// TIA Portal V15.1 export
// export: Created 2020-12-28T13:40:55.3097416Z, ExportSetting WithDefaults, WithReadOnly, DisplayName Totally Integrated Automation Portal, DisplayVersion V15.1 Update 3, DisplayName TIA Portal Openness, DisplayVersion V15.1, DisplayName STEP 7 Professional, DisplayVersion V15.1 Update 3, DisplayName WinCC Advanced, DisplayVersion V15.1 Update 3
DATA_BLOCK "INST TBL TABLE LH"   // DB900
{ S7_Optimized_Access := 'TRUE' }
VERSION : 0.1
// stored: AutoNumber false, CodeModifiedDate 2020-12-28T13:20:36.0178679Z, CompileDate 2020-12-28T13:40:46.9815401Z, CreationDate 2020-12-28T13:20:35.8743592Z, DBAccessibleFromOPCUA true, DownloadWithoutReinit false, InstanceOfName 3STATE_PISTON, InstanceOfNumber 1101, InstanceOfType FB, InterfaceModifiedDate 2020-12-10T07:03:04.0661374Z, IsConsistent true, IsKnowHowProtected false, IsRetainMemResEnabled false, MemoryReserve 100, ModifiedDate 2020-12-28T13:20:36.0178679Z, ParameterModified 2020-12-10T07:03:04.0661374Z, StructureModified 2020-12-10T07:03:04.0661374Z, UDAEnableTagReadback false
"3STATE_PISTON"
   // VAR_INPUT
   //    in_safety : Bool;
   //    in_move_hp : Bool;
   //    in_move_wp : Bool;
   //    in_move_idle : Bool;
   //    in_sensor_hp : Bool;
   //    in_sensor_wp : Bool;
   // END_VAR
   // VAR_OUTPUT
   //    out_in_hp : Bool;
   //    out_in_wp : Bool;
   //    out_idle : Bool;
   //    out_status : Int;
   // END_VAR
   // VAR_IN_OUT
   //    in_ez_hp : Bool;
   //    in_ez_wp : Bool;
   //    in_ez_idle : Bool;
   // END_VAR
   // VAR
   //    "time" : Time;
   //    T : Struct
   //       tt1 : IEC_TIMER;
   //       tt2_hp { S7_SetPoint := 'True'} : IEC_TIMER;
   //       tt3_wp { S7_SetPoint := 'True'} : IEC_TIMER;
   //    END_STRUCT;
   // END_VAR
BEGIN
END_DATA_BLOCK

DATA_BLOCK "INST TBL TABLE RH"   // DB901
{ S7_Optimized_Access := 'TRUE' }
VERSION : 0.1
// stored: AutoNumber false, CodeModifiedDate 2020-12-28T13:20:36.0178679Z, CompileDate 2020-12-28T13:40:46.9815401Z, CreationDate 2020-12-28T13:20:35.8743592Z, DBAccessibleFromOPCUA true, DownloadWithoutReinit false, InstanceOfName 3STATE_PISTON, InstanceOfNumber 1101, InstanceOfType FB, InterfaceModifiedDate 2020-12-10T07:03:04.0661374Z, IsConsistent true, IsKnowHowProtected false, IsRetainMemResEnabled false, MemoryReserve 100, ModifiedDate 2020-12-28T13:20:36.0178679Z, ParameterModified 2020-12-10T07:03:04.0661374Z, StructureModified 2020-12-10T07:03:04.0661374Z, UDAEnableTagReadback false
"3STATE_PISTON"
   // VAR_INPUT
   //    in_safety : Bool;
   //    in_move_hp : Bool;
   //    in_move_wp : Bool;
   //    in_move_idle : Bool;
   //    in_sensor_hp : Bool;
   //    in_sensor_wp : Bool;
   // END_VAR
   // VAR_OUTPUT
   //    out_in_hp : Bool;
   //    out_in_wp : Bool;
   //    out_idle : Bool;
   //    out_status : Int;
   // END_VAR
   // VAR_IN_OUT
   //    in_ez_hp : Bool;
   //    in_ez_wp : Bool;
   //    in_ez_idle : Bool;
   // END_VAR
   // VAR
   //    "time" : Time;
   //    T : Struct
   //       tt1 : IEC_TIMER;
   //       tt2_hp { S7_SetPoint := 'True'} : IEC_TIMER;
   //       tt3_wp { S7_SetPoint := 'True'} : IEC_TIMER;
   //    END_STRUCT;
   // END_VAR
BEGIN
END_DATA_BLOCK

DATA_BLOCK "INST TBL SECTION1"   // DB902
{ S7_Optimized_Access := 'TRUE' }
VERSION : 0.1
// stored: AutoNumber false, CodeModifiedDate 2020-12-28T13:20:36.0178679Z, CompileDate 2020-12-28T13:40:46.9815401Z, CreationDate 2020-12-28T13:20:35.8743592Z, DBAccessibleFromOPCUA true, DownloadWithoutReinit false, InstanceOfName 3STATE_PISTON, InstanceOfNumber 1101, InstanceOfType FB, InterfaceModifiedDate 2020-12-10T07:03:04.0661374Z, IsConsistent true, IsKnowHowProtected false, IsRetainMemResEnabled false, MemoryReserve 100, ModifiedDate 2020-12-28T13:20:36.0178679Z, ParameterModified 2020-12-10T07:03:04.0661374Z, StructureModified 2020-12-10T07:03:04.0661374Z, UDAEnableTagReadback false
"3STATE_PISTON"
   // VAR_INPUT
   //    in_safety : Bool;
   //    in_move_hp : Bool;
   //    in_move_wp : Bool;
   //    in_move_idle : Bool;
   //    in_sensor_hp : Bool;
   //    in_sensor_wp : Bool;
   // END_VAR
   // VAR_OUTPUT
   //    out_in_hp : Bool;
   //    out_in_wp : Bool;
   //    out_idle : Bool;
   //    out_status : Int;
   // END_VAR
   // VAR_IN_OUT
   //    in_ez_hp : Bool;
   //    in_ez_wp : Bool;
   //    in_ez_idle : Bool;
   // END_VAR
   // VAR
   //    "time" : Time;
   //    T : Struct
   //       tt1 : IEC_TIMER;
   //       tt2_hp { S7_SetPoint := 'True'} : IEC_TIMER;
   //       tt3_wp { S7_SetPoint := 'True'} : IEC_TIMER;
   //    END_STRUCT;
   // END_VAR
BEGIN
END_DATA_BLOCK

DATA_BLOCK "INST TBL SECTION2"   // DB903
{ S7_Optimized_Access := 'TRUE' }
VERSION : 0.1
// stored: AutoNumber false, CodeModifiedDate 2020-12-28T13:20:36.0178679Z, CompileDate 2020-12-28T13:40:46.9815401Z, CreationDate 2020-12-28T13:20:35.8743592Z, DBAccessibleFromOPCUA true, DownloadWithoutReinit false, InstanceOfName 3STATE_PISTON, InstanceOfNumber 1101, InstanceOfType FB, InterfaceModifiedDate 2020-12-10T07:03:04.0661374Z, IsConsistent true, IsKnowHowProtected false, IsRetainMemResEnabled false, MemoryReserve 100, ModifiedDate 2020-12-28T13:20:36.0178679Z, ParameterModified 2020-12-10T07:03:04.0661374Z, StructureModified 2020-12-10T07:03:04.0661374Z, UDAEnableTagReadback false
"3STATE_PISTON"
   // VAR_INPUT
   //    in_safety : Bool;
   //    in_move_hp : Bool;
   //    in_move_wp : Bool;
   //    in_move_idle : Bool;
   //    in_sensor_hp : Bool;
   //    in_sensor_wp : Bool;
   // END_VAR
   // VAR_OUTPUT
   //    out_in_hp : Bool;
   //    out_in_wp : Bool;
   //    out_idle : Bool;
   //    out_status : Int;
   // END_VAR
   // VAR_IN_OUT
   //    in_ez_hp : Bool;
   //    in_ez_wp : Bool;
   //    in_ez_idle : Bool;
   // END_VAR
   // VAR
   //    "time" : Time;
   //    T : Struct
   //       tt1 : IEC_TIMER;
   //       tt2_hp { S7_SetPoint := 'True'} : IEC_TIMER;
   //       tt3_wp { S7_SetPoint := 'True'} : IEC_TIMER;
   //    END_STRUCT;
   // END_VAR
BEGIN
END_DATA_BLOCK

DATA_BLOCK "INST TBL SECTION4 LH"   // DB904
{ S7_Optimized_Access := 'TRUE' }
VERSION : 0.1
// stored: AutoNumber false, CodeModifiedDate 2020-12-28T13:20:36.0178679Z, CompileDate 2020-12-28T13:40:46.9815401Z, CreationDate 2020-12-28T13:20:35.8743592Z, DBAccessibleFromOPCUA true, DownloadWithoutReinit false, InstanceOfName 3STATE_PISTON, InstanceOfNumber 1101, InstanceOfType FB, InterfaceModifiedDate 2020-12-10T07:03:04.0661374Z, IsConsistent true, IsKnowHowProtected false, IsRetainMemResEnabled false, MemoryReserve 100, ModifiedDate 2020-12-28T13:20:36.0178679Z, ParameterModified 2020-12-10T07:03:04.0661374Z, StructureModified 2020-12-10T07:03:04.0661374Z, UDAEnableTagReadback false
"3STATE_PISTON"
   // VAR_INPUT
   //    in_safety : Bool;
   //    in_move_hp : Bool;
   //    in_move_wp : Bool;
   //    in_move_idle : Bool;
   //    in_sensor_hp : Bool;
   //    in_sensor_wp : Bool;
   // END_VAR
   // VAR_OUTPUT
   //    out_in_hp : Bool;
   //    out_in_wp : Bool;
   //    out_idle : Bool;
   //    out_status : Int;
   // END_VAR
   // VAR_IN_OUT
   //    in_ez_hp : Bool;
   //    in_ez_wp : Bool;
   //    in_ez_idle : Bool;
   // END_VAR
   // VAR
   //    "time" : Time;
   //    T : Struct
   //       tt1 : IEC_TIMER;
   //       tt2_hp { S7_SetPoint := 'True'} : IEC_TIMER;
   //       tt3_wp { S7_SetPoint := 'True'} : IEC_TIMER;
   //    END_STRUCT;
   // END_VAR
BEGIN
END_DATA_BLOCK

DATA_BLOCK "INST TBL SECTION4 RH"   // DB905
{ S7_Optimized_Access := 'TRUE' }
VERSION : 0.1
// stored: AutoNumber false, CodeModifiedDate 2020-12-28T13:20:36.0178679Z, CompileDate 2020-12-28T13:40:46.9815401Z, CreationDate 2020-12-28T13:20:35.8743592Z, DBAccessibleFromOPCUA true, DownloadWithoutReinit false, InstanceOfName 3STATE_PISTON, InstanceOfNumber 1101, InstanceOfType FB, InterfaceModifiedDate 2020-12-10T07:03:04.0661374Z, IsConsistent true, IsKnowHowProtected false, IsRetainMemResEnabled false, MemoryReserve 100, ModifiedDate 2020-12-28T13:20:36.0178679Z, ParameterModified 2020-12-10T07:03:04.0661374Z, StructureModified 2020-12-10T07:03:04.0661374Z, UDAEnableTagReadback false
"3STATE_PISTON"
   // VAR_INPUT
   //    in_safety : Bool;
   //    in_move_hp : Bool;
   //    in_move_wp : Bool;
   //    in_move_idle : Bool;
   //    in_sensor_hp : Bool;
   //    in_sensor_wp : Bool;
   // END_VAR
   // VAR_OUTPUT
   //    out_in_hp : Bool;
   //    out_in_wp : Bool;
   //    out_idle : Bool;
   //    out_status : Int;
   // END_VAR
   // VAR_IN_OUT
   //    in_ez_hp : Bool;
   //    in_ez_wp : Bool;
   //    in_ez_idle : Bool;
   // END_VAR
   // VAR
   //    "time" : Time;
   //    T : Struct
   //       tt1 : IEC_TIMER;
   //       tt2_hp { S7_SetPoint := 'True'} : IEC_TIMER;
   //       tt3_wp { S7_SetPoint := 'True'} : IEC_TIMER;
   //    END_STRUCT;
   // END_VAR
BEGIN
END_DATA_BLOCK

DATA_BLOCK "INST TBL SECTION5 LH"   // DB906
{ S7_Optimized_Access := 'TRUE' }
VERSION : 0.1
// stored: AutoNumber false, CodeModifiedDate 2020-12-28T13:20:36.0178679Z, CompileDate 2020-12-28T13:40:46.9815401Z, CreationDate 2020-12-28T13:20:35.8743592Z, DBAccessibleFromOPCUA true, DownloadWithoutReinit false, InstanceOfName 3STATE_PISTON, InstanceOfNumber 1101, InstanceOfType FB, InterfaceModifiedDate 2020-12-10T07:03:04.0661374Z, IsConsistent true, IsKnowHowProtected false, IsRetainMemResEnabled false, MemoryReserve 100, ModifiedDate 2020-12-28T13:20:36.0178679Z, ParameterModified 2020-12-10T07:03:04.0661374Z, StructureModified 2020-12-10T07:03:04.0661374Z, UDAEnableTagReadback false
"3STATE_PISTON"
   // VAR_INPUT
   //    in_safety : Bool;
   //    in_move_hp : Bool;
   //    in_move_wp : Bool;
   //    in_move_idle : Bool;
   //    in_sensor_hp : Bool;
   //    in_sensor_wp : Bool;
   // END_VAR
   // VAR_OUTPUT
   //    out_in_hp : Bool;
   //    out_in_wp : Bool;
   //    out_idle : Bool;
   //    out_status : Int;
   // END_VAR
   // VAR_IN_OUT
   //    in_ez_hp : Bool;
   //    in_ez_wp : Bool;
   //    in_ez_idle : Bool;
   // END_VAR
   // VAR
   //    "time" : Time;
   //    T : Struct
   //       tt1 : IEC_TIMER;
   //       tt2_hp { S7_SetPoint := 'True'} : IEC_TIMER;
   //       tt3_wp { S7_SetPoint := 'True'} : IEC_TIMER;
   //    END_STRUCT;
   // END_VAR
BEGIN
END_DATA_BLOCK

DATA_BLOCK "INST TBL SECTION5 RH"   // DB907
{ S7_Optimized_Access := 'TRUE' }
VERSION : 0.1
// stored: AutoNumber false, CodeModifiedDate 2020-12-28T13:20:36.0178679Z, CompileDate 2020-12-28T13:40:46.9815401Z, CreationDate 2020-12-28T13:20:35.8743592Z, DBAccessibleFromOPCUA true, DownloadWithoutReinit false, InstanceOfName 3STATE_PISTON, InstanceOfNumber 1101, InstanceOfType FB, InterfaceModifiedDate 2020-12-10T07:03:04.0661374Z, IsConsistent true, IsKnowHowProtected false, IsRetainMemResEnabled false, MemoryReserve 100, ModifiedDate 2020-12-28T13:20:36.0178679Z, ParameterModified 2020-12-10T07:03:04.0661374Z, StructureModified 2020-12-10T07:03:04.0661374Z, UDAEnableTagReadback false
"3STATE_PISTON"
   // VAR_INPUT
   //    in_safety : Bool;
   //    in_move_hp : Bool;
   //    in_move_wp : Bool;
   //    in_move_idle : Bool;
   //    in_sensor_hp : Bool;
   //    in_sensor_wp : Bool;
   // END_VAR
   // VAR_OUTPUT
   //    out_in_hp : Bool;
   //    out_in_wp : Bool;
   //    out_idle : Bool;
   //    out_status : Int;
   // END_VAR
   // VAR_IN_OUT
   //    in_ez_hp : Bool;
   //    in_ez_wp : Bool;
   //    in_ez_idle : Bool;
   // END_VAR
   // VAR
   //    "time" : Time;
   //    T : Struct
   //       tt1 : IEC_TIMER;
   //       tt2_hp { S7_SetPoint := 'True'} : IEC_TIMER;
   //       tt3_wp { S7_SetPoint := 'True'} : IEC_TIMER;
   //    END_STRUCT;
   // END_VAR
BEGIN
END_DATA_BLOCK

DATA_BLOCK "INST TBL POSITIONING LH"   // DB908
{ S7_Optimized_Access := 'TRUE' }
VERSION : 0.1
// stored: AutoNumber false, CodeModifiedDate 2020-12-28T13:20:36.0178679Z, CompileDate 2020-12-28T13:40:46.9815401Z, CreationDate 2020-12-28T13:20:35.8743592Z, DBAccessibleFromOPCUA true, DownloadWithoutReinit false, InstanceOfName 3STATE_PISTON, InstanceOfNumber 1101, InstanceOfType FB, InterfaceModifiedDate 2020-12-10T07:03:04.0661374Z, IsConsistent true, IsKnowHowProtected false, IsRetainMemResEnabled false, MemoryReserve 100, ModifiedDate 2020-12-28T13:20:36.0178679Z, ParameterModified 2020-12-10T07:03:04.0661374Z, StructureModified 2020-12-10T07:03:04.0661374Z, UDAEnableTagReadback false
"3STATE_PISTON"
   // VAR_INPUT
   //    in_safety : Bool;
   //    in_move_hp : Bool;
   //    in_move_wp : Bool;
   //    in_move_idle : Bool;
   //    in_sensor_hp : Bool;
   //    in_sensor_wp : Bool;
   // END_VAR
   // VAR_OUTPUT
   //    out_in_hp : Bool;
   //    out_in_wp : Bool;
   //    out_idle : Bool;
   //    out_status : Int;
   // END_VAR
   // VAR_IN_OUT
   //    in_ez_hp : Bool;
   //    in_ez_wp : Bool;
   //    in_ez_idle : Bool;
   // END_VAR
   // VAR
   //    "time" : Time;
   //    T : Struct
   //       tt1 : IEC_TIMER;
   //       tt2_hp { S7_SetPoint := 'True'} : IEC_TIMER;
   //       tt3_wp { S7_SetPoint := 'True'} : IEC_TIMER;
   //    END_STRUCT;
   // END_VAR
BEGIN
END_DATA_BLOCK

DATA_BLOCK "INST TBL POSITIONING RH"   // DB909
{ S7_Optimized_Access := 'TRUE' }
VERSION : 0.1
// stored: AutoNumber false, CodeModifiedDate 2020-12-28T13:20:36.0178679Z, CompileDate 2020-12-28T13:40:46.9815401Z, CreationDate 2020-12-28T13:20:35.8743592Z, DBAccessibleFromOPCUA true, DownloadWithoutReinit false, InstanceOfName 3STATE_PISTON, InstanceOfNumber 1101, InstanceOfType FB, InterfaceModifiedDate 2020-12-10T07:03:04.0661374Z, IsConsistent true, IsKnowHowProtected false, IsRetainMemResEnabled false, MemoryReserve 100, ModifiedDate 2020-12-28T13:20:36.0178679Z, ParameterModified 2020-12-10T07:03:04.0661374Z, StructureModified 2020-12-10T07:03:04.0661374Z, UDAEnableTagReadback false
"3STATE_PISTON"
   // VAR_INPUT
   //    in_safety : Bool;
   //    in_move_hp : Bool;
   //    in_move_wp : Bool;
   //    in_move_idle : Bool;
   //    in_sensor_hp : Bool;
   //    in_sensor_wp : Bool;
   // END_VAR
   // VAR_OUTPUT
   //    out_in_hp : Bool;
   //    out_in_wp : Bool;
   //    out_idle : Bool;
   //    out_status : Int;
   // END_VAR
   // VAR_IN_OUT
   //    in_ez_hp : Bool;
   //    in_ez_wp : Bool;
   //    in_ez_idle : Bool;
   // END_VAR
   // VAR
   //    "time" : Time;
   //    T : Struct
   //       tt1 : IEC_TIMER;
   //       tt2_hp { S7_SetPoint := 'True'} : IEC_TIMER;
   //       tt3_wp { S7_SetPoint := 'True'} : IEC_TIMER;
   //    END_STRUCT;
   // END_VAR
BEGIN
END_DATA_BLOCK

DATA_BLOCK "INST TBL PIN LH"   // DB910
{ S7_Optimized_Access := 'TRUE' }
VERSION : 0.1
// stored: AutoNumber false, CodeModifiedDate 2020-12-28T13:20:36.0178679Z, CompileDate 2020-12-28T13:40:46.9815401Z, CreationDate 2020-12-28T13:20:35.8743592Z, DBAccessibleFromOPCUA true, DownloadWithoutReinit false, InstanceOfName 3STATE_PISTON, InstanceOfNumber 1101, InstanceOfType FB, InterfaceModifiedDate 2020-12-10T07:03:04.0661374Z, IsConsistent true, IsKnowHowProtected false, IsRetainMemResEnabled false, MemoryReserve 100, ModifiedDate 2020-12-28T13:20:36.0178679Z, ParameterModified 2020-12-10T07:03:04.0661374Z, StructureModified 2020-12-10T07:03:04.0661374Z, UDAEnableTagReadback false
"3STATE_PISTON"
   // VAR_INPUT
   //    in_safety : Bool;
   //    in_move_hp : Bool;
   //    in_move_wp : Bool;
   //    in_move_idle : Bool;
   //    in_sensor_hp : Bool;
   //    in_sensor_wp : Bool;
   // END_VAR
   // VAR_OUTPUT
   //    out_in_hp : Bool;
   //    out_in_wp : Bool;
   //    out_idle : Bool;
   //    out_status : Int;
   // END_VAR
   // VAR_IN_OUT
   //    in_ez_hp : Bool;
   //    in_ez_wp : Bool;
   //    in_ez_idle : Bool;
   // END_VAR
   // VAR
   //    "time" : Time;
   //    T : Struct
   //       tt1 : IEC_TIMER;
   //       tt2_hp { S7_SetPoint := 'True'} : IEC_TIMER;
   //       tt3_wp { S7_SetPoint := 'True'} : IEC_TIMER;
   //    END_STRUCT;
   // END_VAR
BEGIN
END_DATA_BLOCK

DATA_BLOCK "INST TBL PIN RH"   // DB911
{ S7_Optimized_Access := 'TRUE' }
VERSION : 0.1
// stored: AutoNumber false, CodeModifiedDate 2020-12-28T13:20:36.0178679Z, CompileDate 2020-12-28T13:40:46.9815401Z, CreationDate 2020-12-28T13:20:35.8743592Z, DBAccessibleFromOPCUA true, DownloadWithoutReinit false, InstanceOfName 3STATE_PISTON, InstanceOfNumber 1101, InstanceOfType FB, InterfaceModifiedDate 2020-12-10T07:03:04.0661374Z, IsConsistent true, IsKnowHowProtected false, IsRetainMemResEnabled false, MemoryReserve 100, ModifiedDate 2020-12-28T13:20:36.0178679Z, ParameterModified 2020-12-10T07:03:04.0661374Z, StructureModified 2020-12-10T07:03:04.0661374Z, UDAEnableTagReadback false
"3STATE_PISTON"
   // VAR_INPUT
   //    in_safety : Bool;
   //    in_move_hp : Bool;
   //    in_move_wp : Bool;
   //    in_move_idle : Bool;
   //    in_sensor_hp : Bool;
   //    in_sensor_wp : Bool;
   // END_VAR
   // VAR_OUTPUT
   //    out_in_hp : Bool;
   //    out_in_wp : Bool;
   //    out_idle : Bool;
   //    out_status : Int;
   // END_VAR
   // VAR_IN_OUT
   //    in_ez_hp : Bool;
   //    in_ez_wp : Bool;
   //    in_ez_idle : Bool;
   // END_VAR
   // VAR
   //    "time" : Time;
   //    T : Struct
   //       tt1 : IEC_TIMER;
   //       tt2_hp { S7_SetPoint := 'True'} : IEC_TIMER;
   //       tt3_wp { S7_SetPoint := 'True'} : IEC_TIMER;
   //    END_STRUCT;
   // END_VAR
BEGIN
END_DATA_BLOCK

DATA_BLOCK "INST TBL SCREW GRIPPER"   // DB912
{ S7_Optimized_Access := 'TRUE' }
VERSION : 0.1
// stored: AutoNumber false, CodeModifiedDate 2020-12-28T13:20:36.0178679Z, CompileDate 2020-12-28T13:40:46.9815401Z, CreationDate 2020-12-28T13:20:35.8743592Z, DBAccessibleFromOPCUA true, DownloadWithoutReinit false, InstanceOfName 3STATE_PISTON, InstanceOfNumber 1101, InstanceOfType FB, InterfaceModifiedDate 2020-12-10T07:03:04.0661374Z, IsConsistent true, IsKnowHowProtected false, IsRetainMemResEnabled false, MemoryReserve 100, ModifiedDate 2020-12-28T13:20:36.0178679Z, ParameterModified 2020-12-10T07:03:04.0661374Z, StructureModified 2020-12-10T07:03:04.0661374Z, UDAEnableTagReadback false
"3STATE_PISTON"
   // VAR_INPUT
   //    in_safety : Bool;
   //    in_move_hp : Bool;
   //    in_move_wp : Bool;
   //    in_move_idle : Bool;
   //    in_sensor_hp : Bool;
   //    in_sensor_wp : Bool;
   // END_VAR
   // VAR_OUTPUT
   //    out_in_hp : Bool;
   //    out_in_wp : Bool;
   //    out_idle : Bool;
   //    out_status : Int;
   // END_VAR
   // VAR_IN_OUT
   //    in_ez_hp : Bool;
   //    in_ez_wp : Bool;
   //    in_ez_idle : Bool;
   // END_VAR
   // VAR
   //    "time" : Time;
   //    T : Struct
   //       tt1 : IEC_TIMER;
   //       tt2_hp { S7_SetPoint := 'True'} : IEC_TIMER;
   //       tt3_wp { S7_SetPoint := 'True'} : IEC_TIMER;
   //    END_STRUCT;
   // END_VAR
BEGIN
END_DATA_BLOCK

DATA_BLOCK "INST TBL WRAP GRIPPER"   // DB913
{ S7_Optimized_Access := 'TRUE' }
VERSION : 0.1
// stored: AutoNumber false, CodeModifiedDate 2020-12-28T13:20:36.0178679Z, CompileDate 2020-12-28T13:40:46.9815401Z, CreationDate 2020-12-28T13:20:35.8743592Z, DBAccessibleFromOPCUA true, DownloadWithoutReinit false, InstanceOfName 3STATE_PISTON, InstanceOfNumber 1101, InstanceOfType FB, InterfaceModifiedDate 2020-12-10T07:03:04.0661374Z, IsConsistent true, IsKnowHowProtected false, IsRetainMemResEnabled false, MemoryReserve 100, ModifiedDate 2020-12-28T13:20:36.0178679Z, ParameterModified 2020-12-10T07:03:04.0661374Z, StructureModified 2020-12-10T07:03:04.0661374Z, UDAEnableTagReadback false
"3STATE_PISTON"
   // VAR_INPUT
   //    in_safety : Bool;
   //    in_move_hp : Bool;
   //    in_move_wp : Bool;
   //    in_move_idle : Bool;
   //    in_sensor_hp : Bool;
   //    in_sensor_wp : Bool;
   // END_VAR
   // VAR_OUTPUT
   //    out_in_hp : Bool;
   //    out_in_wp : Bool;
   //    out_idle : Bool;
   //    out_status : Int;
   // END_VAR
   // VAR_IN_OUT
   //    in_ez_hp : Bool;
   //    in_ez_wp : Bool;
   //    in_ez_idle : Bool;
   // END_VAR
   // VAR
   //    "time" : Time;
   //    T : Struct
   //       tt1 : IEC_TIMER;
   //       tt2_hp { S7_SetPoint := 'True'} : IEC_TIMER;
   //       tt3_wp { S7_SetPoint := 'True'} : IEC_TIMER;
   //    END_STRUCT;
   // END_VAR
BEGIN
END_DATA_BLOCK

DATA_BLOCK "INST ST1 POSITIONING"   // DB914
{ S7_Optimized_Access := 'TRUE' }
VERSION : 0.1
// stored: AutoNumber false, CodeModifiedDate 2020-12-28T13:20:36.0178679Z, CompileDate 2020-12-28T13:40:46.9815401Z, CreationDate 2020-12-28T13:20:35.8743592Z, DBAccessibleFromOPCUA true, DownloadWithoutReinit false, InstanceOfName 3STATE_PISTON, InstanceOfNumber 1101, InstanceOfType FB, InterfaceModifiedDate 2020-12-10T07:03:04.0661374Z, IsConsistent true, IsKnowHowProtected false, IsRetainMemResEnabled false, MemoryReserve 100, ModifiedDate 2020-12-28T13:20:36.0178679Z, ParameterModified 2020-12-10T07:03:04.0661374Z, StructureModified 2020-12-10T07:03:04.0661374Z, UDAEnableTagReadback false
"3STATE_PISTON"
   // VAR_INPUT
   //    in_safety : Bool;
   //    in_move_hp : Bool;
   //    in_move_wp : Bool;
   //    in_move_idle : Bool;
   //    in_sensor_hp : Bool;
   //    in_sensor_wp : Bool;
   // END_VAR
   // VAR_OUTPUT
   //    out_in_hp : Bool;
   //    out_in_wp : Bool;
   //    out_idle : Bool;
   //    out_status : Int;
   // END_VAR
   // VAR_IN_OUT
   //    in_ez_hp : Bool;
   //    in_ez_wp : Bool;
   //    in_ez_idle : Bool;
   // END_VAR
   // VAR
   //    "time" : Time;
   //    T : Struct
   //       tt1 : IEC_TIMER;
   //       tt2_hp { S7_SetPoint := 'True'} : IEC_TIMER;
   //       tt3_wp { S7_SetPoint := 'True'} : IEC_TIMER;
   //    END_STRUCT;
   // END_VAR
BEGIN
END_DATA_BLOCK

DATA_BLOCK "INST ST1 SWORD"   // DB915
{ S7_Optimized_Access := 'TRUE' }
VERSION : 0.1
// stored: AutoNumber false, CodeModifiedDate 2020-12-28T13:20:36.0178679Z, CompileDate 2020-12-28T13:40:46.9815401Z, CreationDate 2020-12-28T13:20:35.8743592Z, DBAccessibleFromOPCUA true, DownloadWithoutReinit false, InstanceOfName 3STATE_PISTON, InstanceOfNumber 1101, InstanceOfType FB, InterfaceModifiedDate 2020-12-10T07:03:04.0661374Z, IsConsistent true, IsKnowHowProtected false, IsRetainMemResEnabled false, MemoryReserve 100, ModifiedDate 2020-12-28T13:20:36.0178679Z, ParameterModified 2020-12-10T07:03:04.0661374Z, StructureModified 2020-12-10T07:03:04.0661374Z, UDAEnableTagReadback false
"3STATE_PISTON"
   // VAR_INPUT
   //    in_safety : Bool;
   //    in_move_hp : Bool;
   //    in_move_wp : Bool;
   //    in_move_idle : Bool;
   //    in_sensor_hp : Bool;
   //    in_sensor_wp : Bool;
   // END_VAR
   // VAR_OUTPUT
   //    out_in_hp : Bool;
   //    out_in_wp : Bool;
   //    out_idle : Bool;
   //    out_status : Int;
   // END_VAR
   // VAR_IN_OUT
   //    in_ez_hp : Bool;
   //    in_ez_wp : Bool;
   //    in_ez_idle : Bool;
   // END_VAR
   // VAR
   //    "time" : Time;
   //    T : Struct
   //       tt1 : IEC_TIMER;
   //       tt2_hp { S7_SetPoint := 'True'} : IEC_TIMER;
   //       tt3_wp { S7_SetPoint := 'True'} : IEC_TIMER;
   //    END_STRUCT;
   // END_VAR
BEGIN
END_DATA_BLOCK

DATA_BLOCK "INST ST2 POSITIONING"   // DB916
{ S7_Optimized_Access := 'TRUE' }
VERSION : 0.1
// stored: AutoNumber false, CodeModifiedDate 2020-12-28T13:20:36.0178679Z, CompileDate 2020-12-28T13:40:46.9815401Z, CreationDate 2020-12-28T13:20:35.8743592Z, DBAccessibleFromOPCUA true, DownloadWithoutReinit false, InstanceOfName 3STATE_PISTON, InstanceOfNumber 1101, InstanceOfType FB, InterfaceModifiedDate 2020-12-10T07:03:04.0661374Z, IsConsistent true, IsKnowHowProtected false, IsRetainMemResEnabled false, MemoryReserve 100, ModifiedDate 2020-12-28T13:20:36.0178679Z, ParameterModified 2020-12-10T07:03:04.0661374Z, StructureModified 2020-12-10T07:03:04.0661374Z, UDAEnableTagReadback false
"3STATE_PISTON"
   // VAR_INPUT
   //    in_safety : Bool;
   //    in_move_hp : Bool;
   //    in_move_wp : Bool;
   //    in_move_idle : Bool;
   //    in_sensor_hp : Bool;
   //    in_sensor_wp : Bool;
   // END_VAR
   // VAR_OUTPUT
   //    out_in_hp : Bool;
   //    out_in_wp : Bool;
   //    out_idle : Bool;
   //    out_status : Int;
   // END_VAR
   // VAR_IN_OUT
   //    in_ez_hp : Bool;
   //    in_ez_wp : Bool;
   //    in_ez_idle : Bool;
   // END_VAR
   // VAR
   //    "time" : Time;
   //    T : Struct
   //       tt1 : IEC_TIMER;
   //       tt2_hp { S7_SetPoint := 'True'} : IEC_TIMER;
   //       tt3_wp { S7_SetPoint := 'True'} : IEC_TIMER;
   //    END_STRUCT;
   // END_VAR
BEGIN
END_DATA_BLOCK

DATA_BLOCK "INST ST2 SWORD"   // DB917
{ S7_Optimized_Access := 'TRUE' }
VERSION : 0.1
// stored: AutoNumber false, CodeModifiedDate 2020-12-28T13:20:36.0178679Z, CompileDate 2020-12-28T13:40:46.9815401Z, CreationDate 2020-12-28T13:20:35.8743592Z, DBAccessibleFromOPCUA true, DownloadWithoutReinit false, InstanceOfName 3STATE_PISTON, InstanceOfNumber 1101, InstanceOfType FB, InterfaceModifiedDate 2020-12-10T07:03:04.0661374Z, IsConsistent true, IsKnowHowProtected false, IsRetainMemResEnabled false, MemoryReserve 100, ModifiedDate 2020-12-28T13:20:36.0178679Z, ParameterModified 2020-12-10T07:03:04.0661374Z, StructureModified 2020-12-10T07:03:04.0661374Z, UDAEnableTagReadback false
"3STATE_PISTON"
   // VAR_INPUT
   //    in_safety : Bool;
   //    in_move_hp : Bool;
   //    in_move_wp : Bool;
   //    in_move_idle : Bool;
   //    in_sensor_hp : Bool;
   //    in_sensor_wp : Bool;
   // END_VAR
   // VAR_OUTPUT
   //    out_in_hp : Bool;
   //    out_in_wp : Bool;
   //    out_idle : Bool;
   //    out_status : Int;
   // END_VAR
   // VAR_IN_OUT
   //    in_ez_hp : Bool;
   //    in_ez_wp : Bool;
   //    in_ez_idle : Bool;
   // END_VAR
   // VAR
   //    "time" : Time;
   //    T : Struct
   //       tt1 : IEC_TIMER;
   //       tt2_hp { S7_SetPoint := 'True'} : IEC_TIMER;
   //       tt3_wp { S7_SetPoint := 'True'} : IEC_TIMER;
   //    END_STRUCT;
   // END_VAR
BEGIN
END_DATA_BLOCK

DATA_BLOCK "INST ST3 POSITIONING"   // DB918
{ S7_Optimized_Access := 'TRUE' }
VERSION : 0.1
// stored: AutoNumber false, CodeModifiedDate 2020-12-28T13:20:36.0178679Z, CompileDate 2020-12-28T13:40:46.9815401Z, CreationDate 2020-12-28T13:20:35.8743592Z, DBAccessibleFromOPCUA true, DownloadWithoutReinit false, InstanceOfName 3STATE_PISTON, InstanceOfNumber 1101, InstanceOfType FB, InterfaceModifiedDate 2020-12-10T07:03:04.0661374Z, IsConsistent true, IsKnowHowProtected false, IsRetainMemResEnabled false, MemoryReserve 100, ModifiedDate 2020-12-28T13:20:36.0178679Z, ParameterModified 2020-12-10T07:03:04.0661374Z, StructureModified 2020-12-10T07:03:04.0661374Z, UDAEnableTagReadback false
"3STATE_PISTON"
   // VAR_INPUT
   //    in_safety : Bool;
   //    in_move_hp : Bool;
   //    in_move_wp : Bool;
   //    in_move_idle : Bool;
   //    in_sensor_hp : Bool;
   //    in_sensor_wp : Bool;
   // END_VAR
   // VAR_OUTPUT
   //    out_in_hp : Bool;
   //    out_in_wp : Bool;
   //    out_idle : Bool;
   //    out_status : Int;
   // END_VAR
   // VAR_IN_OUT
   //    in_ez_hp : Bool;
   //    in_ez_wp : Bool;
   //    in_ez_idle : Bool;
   // END_VAR
   // VAR
   //    "time" : Time;
   //    T : Struct
   //       tt1 : IEC_TIMER;
   //       tt2_hp { S7_SetPoint := 'True'} : IEC_TIMER;
   //       tt3_wp { S7_SetPoint := 'True'} : IEC_TIMER;
   //    END_STRUCT;
   // END_VAR
BEGIN
END_DATA_BLOCK

DATA_BLOCK "INST ST3 SWORD A SQUEEZING"   // DB919
{ S7_Optimized_Access := 'TRUE' }
VERSION : 0.1
// stored: AutoNumber false, CodeModifiedDate 2020-12-28T13:20:36.0178679Z, CompileDate 2020-12-28T13:40:46.9815401Z, CreationDate 2020-12-28T13:20:35.8743592Z, DBAccessibleFromOPCUA true, DownloadWithoutReinit false, InstanceOfName 3STATE_PISTON, InstanceOfNumber 1101, InstanceOfType FB, InterfaceModifiedDate 2020-12-10T07:03:04.0661374Z, IsConsistent true, IsKnowHowProtected false, IsRetainMemResEnabled false, MemoryReserve 100, ModifiedDate 2020-12-28T13:20:36.0178679Z, ParameterModified 2020-12-10T07:03:04.0661374Z, StructureModified 2020-12-10T07:03:04.0661374Z, UDAEnableTagReadback false
"3STATE_PISTON"
   // VAR_INPUT
   //    in_safety : Bool;
   //    in_move_hp : Bool;
   //    in_move_wp : Bool;
   //    in_move_idle : Bool;
   //    in_sensor_hp : Bool;
   //    in_sensor_wp : Bool;
   // END_VAR
   // VAR_OUTPUT
   //    out_in_hp : Bool;
   //    out_in_wp : Bool;
   //    out_idle : Bool;
   //    out_status : Int;
   // END_VAR
   // VAR_IN_OUT
   //    in_ez_hp : Bool;
   //    in_ez_wp : Bool;
   //    in_ez_idle : Bool;
   // END_VAR
   // VAR
   //    "time" : Time;
   //    T : Struct
   //       tt1 : IEC_TIMER;
   //       tt2_hp { S7_SetPoint := 'True'} : IEC_TIMER;
   //       tt3_wp { S7_SetPoint := 'True'} : IEC_TIMER;
   //    END_STRUCT;
   // END_VAR
BEGIN
END_DATA_BLOCK

DATA_BLOCK "INST ST3 SWORD A SPREADING"   // DB920
{ S7_Optimized_Access := 'TRUE' }
VERSION : 0.1
// stored: AutoNumber false, CodeModifiedDate 2020-12-28T13:20:36.0178679Z, CompileDate 2020-12-28T13:40:46.9815401Z, CreationDate 2020-12-28T13:20:35.8743592Z, DBAccessibleFromOPCUA true, DownloadWithoutReinit false, InstanceOfName 3STATE_PISTON, InstanceOfNumber 1101, InstanceOfType FB, InterfaceModifiedDate 2020-12-10T07:03:04.0661374Z, IsConsistent true, IsKnowHowProtected false, IsRetainMemResEnabled false, MemoryReserve 100, ModifiedDate 2020-12-28T13:20:36.0178679Z, ParameterModified 2020-12-10T07:03:04.0661374Z, StructureModified 2020-12-10T07:03:04.0661374Z, UDAEnableTagReadback false
"3STATE_PISTON"
   // VAR_INPUT
   //    in_safety : Bool;
   //    in_move_hp : Bool;
   //    in_move_wp : Bool;
   //    in_move_idle : Bool;
   //    in_sensor_hp : Bool;
   //    in_sensor_wp : Bool;
   // END_VAR
   // VAR_OUTPUT
   //    out_in_hp : Bool;
   //    out_in_wp : Bool;
   //    out_idle : Bool;
   //    out_status : Int;
   // END_VAR
   // VAR_IN_OUT
   //    in_ez_hp : Bool;
   //    in_ez_wp : Bool;
   //    in_ez_idle : Bool;
   // END_VAR
   // VAR
   //    "time" : Time;
   //    T : Struct
   //       tt1 : IEC_TIMER;
   //       tt2_hp { S7_SetPoint := 'True'} : IEC_TIMER;
   //       tt3_wp { S7_SetPoint := 'True'} : IEC_TIMER;
   //    END_STRUCT;
   // END_VAR
BEGIN
END_DATA_BLOCK

DATA_BLOCK "INST ST3 SWORD A OPENING"   // DB921
{ S7_Optimized_Access := 'TRUE' }
VERSION : 0.1
// stored: AutoNumber false, CodeModifiedDate 2020-12-28T13:20:36.0178679Z, CompileDate 2020-12-28T13:40:46.9815401Z, CreationDate 2020-12-28T13:20:35.8743592Z, DBAccessibleFromOPCUA true, DownloadWithoutReinit false, InstanceOfName 3STATE_PISTON, InstanceOfNumber 1101, InstanceOfType FB, InterfaceModifiedDate 2020-12-10T07:03:04.0661374Z, IsConsistent true, IsKnowHowProtected false, IsRetainMemResEnabled false, MemoryReserve 100, ModifiedDate 2020-12-28T13:20:36.0178679Z, ParameterModified 2020-12-10T07:03:04.0661374Z, StructureModified 2020-12-10T07:03:04.0661374Z, UDAEnableTagReadback false
"3STATE_PISTON"
   // VAR_INPUT
   //    in_safety : Bool;
   //    in_move_hp : Bool;
   //    in_move_wp : Bool;
   //    in_move_idle : Bool;
   //    in_sensor_hp : Bool;
   //    in_sensor_wp : Bool;
   // END_VAR
   // VAR_OUTPUT
   //    out_in_hp : Bool;
   //    out_in_wp : Bool;
   //    out_idle : Bool;
   //    out_status : Int;
   // END_VAR
   // VAR_IN_OUT
   //    in_ez_hp : Bool;
   //    in_ez_wp : Bool;
   //    in_ez_idle : Bool;
   // END_VAR
   // VAR
   //    "time" : Time;
   //    T : Struct
   //       tt1 : IEC_TIMER;
   //       tt2_hp { S7_SetPoint := 'True'} : IEC_TIMER;
   //       tt3_wp { S7_SetPoint := 'True'} : IEC_TIMER;
   //    END_STRUCT;
   // END_VAR
BEGIN
END_DATA_BLOCK

DATA_BLOCK "INST ST3 SWORD B SQUEEZING"   // DB922
{ S7_Optimized_Access := 'TRUE' }
VERSION : 0.1
// stored: AutoNumber false, CodeModifiedDate 2020-12-28T13:20:36.0178679Z, CompileDate 2020-12-28T13:40:46.9815401Z, CreationDate 2020-12-28T13:20:35.8743592Z, DBAccessibleFromOPCUA true, DownloadWithoutReinit false, InstanceOfName 3STATE_PISTON, InstanceOfNumber 1101, InstanceOfType FB, InterfaceModifiedDate 2020-12-10T07:03:04.0661374Z, IsConsistent true, IsKnowHowProtected false, IsRetainMemResEnabled false, MemoryReserve 100, ModifiedDate 2020-12-28T13:20:36.0178679Z, ParameterModified 2020-12-10T07:03:04.0661374Z, StructureModified 2020-12-10T07:03:04.0661374Z, UDAEnableTagReadback false
"3STATE_PISTON"
   // VAR_INPUT
   //    in_safety : Bool;
   //    in_move_hp : Bool;
   //    in_move_wp : Bool;
   //    in_move_idle : Bool;
   //    in_sensor_hp : Bool;
   //    in_sensor_wp : Bool;
   // END_VAR
   // VAR_OUTPUT
   //    out_in_hp : Bool;
   //    out_in_wp : Bool;
   //    out_idle : Bool;
   //    out_status : Int;
   // END_VAR
   // VAR_IN_OUT
   //    in_ez_hp : Bool;
   //    in_ez_wp : Bool;
   //    in_ez_idle : Bool;
   // END_VAR
   // VAR
   //    "time" : Time;
   //    T : Struct
   //       tt1 : IEC_TIMER;
   //       tt2_hp { S7_SetPoint := 'True'} : IEC_TIMER;
   //       tt3_wp { S7_SetPoint := 'True'} : IEC_TIMER;
   //    END_STRUCT;
   // END_VAR
BEGIN
END_DATA_BLOCK

DATA_BLOCK "INST ST3 SWORD B SPREADING"   // DB923
{ S7_Optimized_Access := 'TRUE' }
VERSION : 0.1
// stored: AutoNumber false, CodeModifiedDate 2020-12-28T13:20:36.0178679Z, CompileDate 2020-12-28T13:40:46.9815401Z, CreationDate 2020-12-28T13:20:35.8743592Z, DBAccessibleFromOPCUA true, DownloadWithoutReinit false, InstanceOfName 3STATE_PISTON, InstanceOfNumber 1101, InstanceOfType FB, InterfaceModifiedDate 2020-12-10T07:03:04.0661374Z, IsConsistent true, IsKnowHowProtected false, IsRetainMemResEnabled false, MemoryReserve 100, ModifiedDate 2020-12-28T13:20:36.0178679Z, ParameterModified 2020-12-10T07:03:04.0661374Z, StructureModified 2020-12-10T07:03:04.0661374Z, UDAEnableTagReadback false
"3STATE_PISTON"
   // VAR_INPUT
   //    in_safety : Bool;
   //    in_move_hp : Bool;
   //    in_move_wp : Bool;
   //    in_move_idle : Bool;
   //    in_sensor_hp : Bool;
   //    in_sensor_wp : Bool;
   // END_VAR
   // VAR_OUTPUT
   //    out_in_hp : Bool;
   //    out_in_wp : Bool;
   //    out_idle : Bool;
   //    out_status : Int;
   // END_VAR
   // VAR_IN_OUT
   //    in_ez_hp : Bool;
   //    in_ez_wp : Bool;
   //    in_ez_idle : Bool;
   // END_VAR
   // VAR
   //    "time" : Time;
   //    T : Struct
   //       tt1 : IEC_TIMER;
   //       tt2_hp { S7_SetPoint := 'True'} : IEC_TIMER;
   //       tt3_wp { S7_SetPoint := 'True'} : IEC_TIMER;
   //    END_STRUCT;
   // END_VAR
BEGIN
END_DATA_BLOCK

DATA_BLOCK "INST ST3 SWORD B OPENING"   // DB924
{ S7_Optimized_Access := 'TRUE' }
VERSION : 0.1
// stored: AutoNumber false, CodeModifiedDate 2020-12-28T13:20:36.0178679Z, CompileDate 2020-12-28T13:40:46.9815401Z, CreationDate 2020-12-28T13:20:35.8743592Z, DBAccessibleFromOPCUA true, DownloadWithoutReinit false, InstanceOfName 3STATE_PISTON, InstanceOfNumber 1101, InstanceOfType FB, InterfaceModifiedDate 2020-12-10T07:03:04.0661374Z, IsConsistent true, IsKnowHowProtected false, IsRetainMemResEnabled false, MemoryReserve 100, ModifiedDate 2020-12-28T13:20:36.0178679Z, ParameterModified 2020-12-10T07:03:04.0661374Z, StructureModified 2020-12-10T07:03:04.0661374Z, UDAEnableTagReadback false
"3STATE_PISTON"
   // VAR_INPUT
   //    in_safety : Bool;
   //    in_move_hp : Bool;
   //    in_move_wp : Bool;
   //    in_move_idle : Bool;
   //    in_sensor_hp : Bool;
   //    in_sensor_wp : Bool;
   // END_VAR
   // VAR_OUTPUT
   //    out_in_hp : Bool;
   //    out_in_wp : Bool;
   //    out_idle : Bool;
   //    out_status : Int;
   // END_VAR
   // VAR_IN_OUT
   //    in_ez_hp : Bool;
   //    in_ez_wp : Bool;
   //    in_ez_idle : Bool;
   // END_VAR
   // VAR
   //    "time" : Time;
   //    T : Struct
   //       tt1 : IEC_TIMER;
   //       tt2_hp { S7_SetPoint := 'True'} : IEC_TIMER;
   //       tt3_wp { S7_SetPoint := 'True'} : IEC_TIMER;
   //    END_STRUCT;
   // END_VAR
BEGIN
END_DATA_BLOCK

DATA_BLOCK "INST ST6 CONNECTOR1"   // DB925
{ S7_Optimized_Access := 'TRUE' }
VERSION : 0.1
// stored: AutoNumber false, CodeModifiedDate 2020-12-28T13:20:36.0178679Z, CompileDate 2020-12-28T13:40:46.9815401Z, CreationDate 2020-12-28T13:20:35.8743592Z, DBAccessibleFromOPCUA true, DownloadWithoutReinit false, InstanceOfName 3STATE_PISTON, InstanceOfNumber 1101, InstanceOfType FB, InterfaceModifiedDate 2020-12-10T07:03:04.0661374Z, IsConsistent true, IsKnowHowProtected false, IsRetainMemResEnabled false, MemoryReserve 100, ModifiedDate 2020-12-28T13:20:36.0178679Z, ParameterModified 2020-12-10T07:03:04.0661374Z, StructureModified 2020-12-10T07:03:04.0661374Z, UDAEnableTagReadback false
"3STATE_PISTON"
   // VAR_INPUT
   //    in_safety : Bool;
   //    in_move_hp : Bool;
   //    in_move_wp : Bool;
   //    in_move_idle : Bool;
   //    in_sensor_hp : Bool;
   //    in_sensor_wp : Bool;
   // END_VAR
   // VAR_OUTPUT
   //    out_in_hp : Bool;
   //    out_in_wp : Bool;
   //    out_idle : Bool;
   //    out_status : Int;
   // END_VAR
   // VAR_IN_OUT
   //    in_ez_hp : Bool;
   //    in_ez_wp : Bool;
   //    in_ez_idle : Bool;
   // END_VAR
   // VAR
   //    "time" : Time;
   //    T : Struct
   //       tt1 : IEC_TIMER;
   //       tt2_hp { S7_SetPoint := 'True'} : IEC_TIMER;
   //       tt3_wp { S7_SetPoint := 'True'} : IEC_TIMER;
   //    END_STRUCT;
   // END_VAR
BEGIN
END_DATA_BLOCK

DATA_BLOCK "INST ST6 CONNECTOR2"   // DB926
{ S7_Optimized_Access := 'TRUE' }
VERSION : 0.1
// stored: AutoNumber false, CodeModifiedDate 2020-12-28T13:20:36.0178679Z, CompileDate 2020-12-28T13:40:46.9815401Z, CreationDate 2020-12-28T13:20:35.8743592Z, DBAccessibleFromOPCUA true, DownloadWithoutReinit false, InstanceOfName 3STATE_PISTON, InstanceOfNumber 1101, InstanceOfType FB, InterfaceModifiedDate 2020-12-10T07:03:04.0661374Z, IsConsistent true, IsKnowHowProtected false, IsRetainMemResEnabled false, MemoryReserve 100, ModifiedDate 2020-12-28T13:20:36.0178679Z, ParameterModified 2020-12-10T07:03:04.0661374Z, StructureModified 2020-12-10T07:03:04.0661374Z, UDAEnableTagReadback false
"3STATE_PISTON"
   // VAR_INPUT
   //    in_safety : Bool;
   //    in_move_hp : Bool;
   //    in_move_wp : Bool;
   //    in_move_idle : Bool;
   //    in_sensor_hp : Bool;
   //    in_sensor_wp : Bool;
   // END_VAR
   // VAR_OUTPUT
   //    out_in_hp : Bool;
   //    out_in_wp : Bool;
   //    out_idle : Bool;
   //    out_status : Int;
   // END_VAR
   // VAR_IN_OUT
   //    in_ez_hp : Bool;
   //    in_ez_wp : Bool;
   //    in_ez_idle : Bool;
   // END_VAR
   // VAR
   //    "time" : Time;
   //    T : Struct
   //       tt1 : IEC_TIMER;
   //       tt2_hp { S7_SetPoint := 'True'} : IEC_TIMER;
   //       tt3_wp { S7_SetPoint := 'True'} : IEC_TIMER;
   //    END_STRUCT;
   // END_VAR
BEGIN
END_DATA_BLOCK

DATA_BLOCK "INST ST6 HOLDFAST LH1"   // DB927
{ S7_Optimized_Access := 'TRUE' }
VERSION : 0.1
// stored: AutoNumber false, CodeModifiedDate 2020-12-28T13:20:36.0178679Z, CompileDate 2020-12-28T13:40:46.9815401Z, CreationDate 2020-12-28T13:20:35.8743592Z, DBAccessibleFromOPCUA true, DownloadWithoutReinit false, InstanceOfName 3STATE_PISTON, InstanceOfNumber 1101, InstanceOfType FB, InterfaceModifiedDate 2020-12-10T07:03:04.0661374Z, IsConsistent true, IsKnowHowProtected false, IsRetainMemResEnabled false, MemoryReserve 100, ModifiedDate 2020-12-28T13:20:36.0178679Z, ParameterModified 2020-12-10T07:03:04.0661374Z, StructureModified 2020-12-10T07:03:04.0661374Z, UDAEnableTagReadback false
"3STATE_PISTON"
   // VAR_INPUT
   //    in_safety : Bool;
   //    in_move_hp : Bool;
   //    in_move_wp : Bool;
   //    in_move_idle : Bool;
   //    in_sensor_hp : Bool;
   //    in_sensor_wp : Bool;
   // END_VAR
   // VAR_OUTPUT
   //    out_in_hp : Bool;
   //    out_in_wp : Bool;
   //    out_idle : Bool;
   //    out_status : Int;
   // END_VAR
   // VAR_IN_OUT
   //    in_ez_hp : Bool;
   //    in_ez_wp : Bool;
   //    in_ez_idle : Bool;
   // END_VAR
   // VAR
   //    "time" : Time;
   //    T : Struct
   //       tt1 : IEC_TIMER;
   //       tt2_hp { S7_SetPoint := 'True'} : IEC_TIMER;
   //       tt3_wp { S7_SetPoint := 'True'} : IEC_TIMER;
   //    END_STRUCT;
   // END_VAR
BEGIN
END_DATA_BLOCK

DATA_BLOCK "INST ST6 HOLDFAST LH2"   // DB928
{ S7_Optimized_Access := 'TRUE' }
VERSION : 0.1
// stored: AutoNumber false, CodeModifiedDate 2020-12-28T13:20:36.0178679Z, CompileDate 2020-12-28T13:40:46.9815401Z, CreationDate 2020-12-28T13:20:35.8743592Z, DBAccessibleFromOPCUA true, DownloadWithoutReinit false, InstanceOfName 3STATE_PISTON, InstanceOfNumber 1101, InstanceOfType FB, InterfaceModifiedDate 2020-12-10T07:03:04.0661374Z, IsConsistent true, IsKnowHowProtected false, IsRetainMemResEnabled false, MemoryReserve 100, ModifiedDate 2020-12-28T13:20:36.0178679Z, ParameterModified 2020-12-10T07:03:04.0661374Z, StructureModified 2020-12-10T07:03:04.0661374Z, UDAEnableTagReadback false
"3STATE_PISTON"
   // VAR_INPUT
   //    in_safety : Bool;
   //    in_move_hp : Bool;
   //    in_move_wp : Bool;
   //    in_move_idle : Bool;
   //    in_sensor_hp : Bool;
   //    in_sensor_wp : Bool;
   // END_VAR
   // VAR_OUTPUT
   //    out_in_hp : Bool;
   //    out_in_wp : Bool;
   //    out_idle : Bool;
   //    out_status : Int;
   // END_VAR
   // VAR_IN_OUT
   //    in_ez_hp : Bool;
   //    in_ez_wp : Bool;
   //    in_ez_idle : Bool;
   // END_VAR
   // VAR
   //    "time" : Time;
   //    T : Struct
   //       tt1 : IEC_TIMER;
   //       tt2_hp { S7_SetPoint := 'True'} : IEC_TIMER;
   //       tt3_wp { S7_SetPoint := 'True'} : IEC_TIMER;
   //    END_STRUCT;
   // END_VAR
BEGIN
END_DATA_BLOCK

DATA_BLOCK "INST ST6 HOLDFAST RH1"   // DB929
{ S7_Optimized_Access := 'TRUE' }
VERSION : 0.1
// stored: AutoNumber false, CodeModifiedDate 2020-12-28T13:20:36.0178679Z, CompileDate 2020-12-28T13:40:46.9815401Z, CreationDate 2020-12-28T13:20:35.8743592Z, DBAccessibleFromOPCUA true, DownloadWithoutReinit false, InstanceOfName 3STATE_PISTON, InstanceOfNumber 1101, InstanceOfType FB, InterfaceModifiedDate 2020-12-10T07:03:04.0661374Z, IsConsistent true, IsKnowHowProtected false, IsRetainMemResEnabled false, MemoryReserve 100, ModifiedDate 2020-12-28T13:20:36.0178679Z, ParameterModified 2020-12-10T07:03:04.0661374Z, StructureModified 2020-12-10T07:03:04.0661374Z, UDAEnableTagReadback false
"3STATE_PISTON"
   // VAR_INPUT
   //    in_safety : Bool;
   //    in_move_hp : Bool;
   //    in_move_wp : Bool;
   //    in_move_idle : Bool;
   //    in_sensor_hp : Bool;
   //    in_sensor_wp : Bool;
   // END_VAR
   // VAR_OUTPUT
   //    out_in_hp : Bool;
   //    out_in_wp : Bool;
   //    out_idle : Bool;
   //    out_status : Int;
   // END_VAR
   // VAR_IN_OUT
   //    in_ez_hp : Bool;
   //    in_ez_wp : Bool;
   //    in_ez_idle : Bool;
   // END_VAR
   // VAR
   //    "time" : Time;
   //    T : Struct
   //       tt1 : IEC_TIMER;
   //       tt2_hp { S7_SetPoint := 'True'} : IEC_TIMER;
   //       tt3_wp { S7_SetPoint := 'True'} : IEC_TIMER;
   //    END_STRUCT;
   // END_VAR
BEGIN
END_DATA_BLOCK

DATA_BLOCK "INST ST6 HOLDFAST RH2"   // DB930
{ S7_Optimized_Access := 'TRUE' }
VERSION : 0.1
// stored: AutoNumber false, CodeModifiedDate 2020-12-28T13:20:36.0178679Z, CompileDate 2020-12-28T13:40:46.9815401Z, CreationDate 2020-12-28T13:20:35.8743592Z, DBAccessibleFromOPCUA true, DownloadWithoutReinit false, InstanceOfName 3STATE_PISTON, InstanceOfNumber 1101, InstanceOfType FB, InterfaceModifiedDate 2020-12-10T07:03:04.0661374Z, IsConsistent true, IsKnowHowProtected false, IsRetainMemResEnabled false, MemoryReserve 100, ModifiedDate 2020-12-28T13:20:36.0178679Z, ParameterModified 2020-12-10T07:03:04.0661374Z, StructureModified 2020-12-10T07:03:04.0661374Z, UDAEnableTagReadback false
"3STATE_PISTON"
   // VAR_INPUT
   //    in_safety : Bool;
   //    in_move_hp : Bool;
   //    in_move_wp : Bool;
   //    in_move_idle : Bool;
   //    in_sensor_hp : Bool;
   //    in_sensor_wp : Bool;
   // END_VAR
   // VAR_OUTPUT
   //    out_in_hp : Bool;
   //    out_in_wp : Bool;
   //    out_idle : Bool;
   //    out_status : Int;
   // END_VAR
   // VAR_IN_OUT
   //    in_ez_hp : Bool;
   //    in_ez_wp : Bool;
   //    in_ez_idle : Bool;
   // END_VAR
   // VAR
   //    "time" : Time;
   //    T : Struct
   //       tt1 : IEC_TIMER;
   //       tt2_hp { S7_SetPoint := 'True'} : IEC_TIMER;
   //       tt3_wp { S7_SetPoint := 'True'} : IEC_TIMER;
   //    END_STRUCT;
   // END_VAR
BEGIN
END_DATA_BLOCK

DATA_BLOCK "INST ST6 ROTATION LH"   // DB931
{ S7_Optimized_Access := 'TRUE' }
VERSION : 0.1
// stored: AutoNumber false, CodeModifiedDate 2020-12-28T13:20:36.0178679Z, CompileDate 2020-12-28T13:40:46.9815401Z, CreationDate 2020-12-28T13:20:35.8743592Z, DBAccessibleFromOPCUA true, DownloadWithoutReinit false, InstanceOfName 3STATE_PISTON, InstanceOfNumber 1101, InstanceOfType FB, InterfaceModifiedDate 2020-12-10T07:03:04.0661374Z, IsConsistent true, IsKnowHowProtected false, IsRetainMemResEnabled false, MemoryReserve 100, ModifiedDate 2020-12-28T13:20:36.0178679Z, ParameterModified 2020-12-10T07:03:04.0661374Z, StructureModified 2020-12-10T07:03:04.0661374Z, UDAEnableTagReadback false
"3STATE_PISTON"
   // VAR_INPUT
   //    in_safety : Bool;
   //    in_move_hp : Bool;
   //    in_move_wp : Bool;
   //    in_move_idle : Bool;
   //    in_sensor_hp : Bool;
   //    in_sensor_wp : Bool;
   // END_VAR
   // VAR_OUTPUT
   //    out_in_hp : Bool;
   //    out_in_wp : Bool;
   //    out_idle : Bool;
   //    out_status : Int;
   // END_VAR
   // VAR_IN_OUT
   //    in_ez_hp : Bool;
   //    in_ez_wp : Bool;
   //    in_ez_idle : Bool;
   // END_VAR
   // VAR
   //    "time" : Time;
   //    T : Struct
   //       tt1 : IEC_TIMER;
   //       tt2_hp { S7_SetPoint := 'True'} : IEC_TIMER;
   //       tt3_wp { S7_SetPoint := 'True'} : IEC_TIMER;
   //    END_STRUCT;
   // END_VAR
BEGIN
END_DATA_BLOCK

DATA_BLOCK "INST ST6 ROTATION RH"   // DB932
{ S7_Optimized_Access := 'TRUE' }
VERSION : 0.1
// stored: AutoNumber false, CodeModifiedDate 2020-12-28T13:20:36.0178679Z, CompileDate 2020-12-28T13:40:46.9815401Z, CreationDate 2020-12-28T13:20:35.8743592Z, DBAccessibleFromOPCUA true, DownloadWithoutReinit false, InstanceOfName 3STATE_PISTON, InstanceOfNumber 1101, InstanceOfType FB, InterfaceModifiedDate 2020-12-10T07:03:04.0661374Z, IsConsistent true, IsKnowHowProtected false, IsRetainMemResEnabled false, MemoryReserve 100, ModifiedDate 2020-12-28T13:20:36.0178679Z, ParameterModified 2020-12-10T07:03:04.0661374Z, StructureModified 2020-12-10T07:03:04.0661374Z, UDAEnableTagReadback false
"3STATE_PISTON"
   // VAR_INPUT
   //    in_safety : Bool;
   //    in_move_hp : Bool;
   //    in_move_wp : Bool;
   //    in_move_idle : Bool;
   //    in_sensor_hp : Bool;
   //    in_sensor_wp : Bool;
   // END_VAR
   // VAR_OUTPUT
   //    out_in_hp : Bool;
   //    out_in_wp : Bool;
   //    out_idle : Bool;
   //    out_status : Int;
   // END_VAR
   // VAR_IN_OUT
   //    in_ez_hp : Bool;
   //    in_ez_wp : Bool;
   //    in_ez_idle : Bool;
   // END_VAR
   // VAR
   //    "time" : Time;
   //    T : Struct
   //       tt1 : IEC_TIMER;
   //       tt2_hp { S7_SetPoint := 'True'} : IEC_TIMER;
   //       tt3_wp { S7_SetPoint := 'True'} : IEC_TIMER;
   //    END_STRUCT;
   // END_VAR
BEGIN
END_DATA_BLOCK
